// TIA Portal V19 export
FUNCTION_BLOCK "Pu_Entl.GP0x"   // FB1009, LAD
TITLE = Pumpe Abpumpen Sump
{ S7_Optimized_Access := 'TRUE' }
// Funktionen:  Entleeren /  Spülen
// stored: AutoNumber false, MemoryReserve 100, SetENOAutomatically false
   VAR RETAIN
      In { ExternalAccessible := 'False'; ExternalVisible := 'False'; ExternalWritable := 'False'} : Struct
         Auto : Bool;   // Paneltaste
         Ein : Bool;   // Paneltaste
         Leckage_ok : Bool;
         Frg_Niv_CM05 : Bool;
         Betriebsart : USInt := 0;   // Paneltaste
      END_STRUCT;
      Param { ExternalAccessible := 'False'; ExternalVisible := 'False'; ExternalWritable := 'False'} : Struct
         Spülzeit : Time;
      END_STRUCT;
      Zst { ExternalAccessible := 'False'; ExternalVisible := 'False'; ExternalWritable := 'False'} : Struct
         Niveau : USInt;
         Status_GP0x : USInt;
         Restzeit_Spülen : Time;
         TON_Spülventil_auf : Bool;
         Spuelen : Bool;
         Abpumpen : Bool;
         Bedienung_Erlaubt : Bool;
      END_STRUCT;
      Mld { ExternalAccessible := 'False'; ExternalVisible := 'False'; ExternalWritable := 'False'} : Struct
         Leckage : Bool;
         Niv_Sensorfehler : Bool;
         n_Auto : Bool;
      END_STRUCT;
      Out { ExternalAccessible := 'False'; ExternalVisible := 'False'; ExternalWritable := 'False'} : Struct
         GP0x_Ein : Bool;
         Spülventil : Bool;
      END_STRUCT;
   END_VAR
   VAR
      IEC_Timer { ExternalAccessible := 'False'; ExternalVisible := 'False'; ExternalWritable := 'False'} : Struct
         Leckage_ok { S7_SetPoint := 'True'} : TON_TIME;
         Spülventil_auf { S7_SetPoint := 'True'} : TON_TIME;
         Spülen { S7_SetPoint := 'True'} : TP_TIME;
         Leckage_niO { S7_SetPoint := 'True'} : TON_TIME;
      END_STRUCT;
      R_TRIG_Hand_EIN { ExternalAccessible := 'False'; ExternalVisible := 'False'; ExternalWritable := 'False'} : R_TRIG;
   END_VAR
   VAR_TEMP
      Spülzeit : Time;
      Leckage_ok_verz : Bool;
      posFl_Hand : Bool;
   END_VAR
   VAR CONSTANT
      Niv_TLS : USInt := 2;
      Niv_Min : USInt := 2;
      Niv_max : USInt := 20;
      Zeit_Ventil_auf : Time := T#1s;
   END_VAR
BEGIN

REGION Network 1 (SCL): Input
   // Panelbedienung und Sensoren --> Input()
   // Leckage o.k. verzögert
   #IEC_Timer.Leckage_ok(IN := #In.Leckage_ok,
                         PT := T#120s,
                         Q => #Leckage_ok_verz);

   // Timer Spülventil AUF
   #IEC_Timer.Spülventil_auf(IN := #Out.Spülventil,
                              PT := #Zeit_Ventil_auf,
                              Q => #Zst.TON_Spülventil_auf);

    // positive Flanke "Hand Ein"
   #R_TRIG_Hand_EIN(CLK := #In.Ein,
                    Q => #posFl_Hand);

   #IEC_Timer.Spülen(IN := #posFl_Hand AND #In.Betriebsart = 1,
                     PT := #Param.Spülzeit,
                     Q => #Zst.Spuelen,
                     ET => #Spülzeit);
END_REGION

REGION Network 2 (SCL): Ansteuerung
   // Zielbehälter nicht voll
   IF #In.Frg_Niv_CM05 THEN
       CASE #In.Betriebsart OF
           0:  // Entleeren

               // Spülventil zu
               #Out.Spülventil := FALSE;
               #Zst.Restzeit_Spülen := T#0s;

               // Wenn Leckage oder einmalig per Hand
               IF #In.Auto AND NOT #In.Leckage_ok OR #posFl_Hand THEN
                   #Zst.Abpumpen := TRUE;
               ELSIF #Leckage_ok_verz THEN
                   #Zst.Abpumpen := FALSE;
               END_IF;

           1: // Spülen - nur Hand
               IF #In.Ein THEN
                   IF #posFl_Hand THEN
                       #Out.Spülventil := TRUE;
                   ELSIF NOT #Zst.Spuelen AND #Zst.TON_Spülventil_auf THEN
                       #Out.Spülventil := FALSE;
                   END_IF;
                   #Zst.Restzeit_Spülen := #Param.Spülzeit - #Spülzeit;
               ELSE
                   #Zst.Spuelen := FALSE;
                   #Out.Spülventil := FALSE;
                   #Zst.Restzeit_Spülen := T#0s;
               END_IF;

               // Wenn Leckage 
               IF #Leckage_ok_verz OR (NOT #In.Auto AND NOT #In.Ein) THEN
                   #Zst.Abpumpen := FALSE;
               ELSIF NOT #In.Leckage_ok THEN
                   #Zst.Abpumpen := TRUE;
               END_IF;
       END_CASE;

       // Pumpe an    
       #Out.GP0x_Ein := #Zst.Abpumpen AND (#In.Auto OR #In.Ein);
   ELSE
       #Out.Spülventil := FALSE;
       #Zst.Restzeit_Spülen := T#0s;
       #Out.GP0x_Ein := FALSE;
   END_IF;
END_REGION

REGION Network 3 (SCL): Überwachung / Meldungen

   // Meldung Leckage verzögert
   #IEC_Timer.Leckage_niO(IN := NOT #In.Leckage_ok,
                   PT := T#30s,
                   Q => #Mld.Leckage);

   // nicht in Automatik
   #Mld.n_Auto := NOT #In.Auto AND "DB_ANLAGE".BA.Automat_ein;
END_REGION

REGION Network 4 (SCL): --> Visu
   // Status Pumpe
   "Status_E0A"(Hand := #In.Ein,
                Auto := #In.Auto,
                SonderModus_PumpeSpuelen:=FALSE,
                Stoerung := FALSE,
                Ausgang := #Out.GP0x_Ein,
                StatusByte => #Zst.Status_GP0x);
   // Anzeige Füllstand
   "Niv_Visu"(Niv_1 := TRUE,
              Niv_2 := NOT #In.Leckage_ok,
              Niv_3 := FALSE,
              Niv_4 := FALSE,
              Niv_5 := FALSE,
              Niv_6 := FALSE,
              Wert_1 := #Niv_Min,
              Wert_2 := #Niv_max,
              Wert_3 := 0,
              Wert_4 := 0,
              Wert_5 := 0,
              Wert_6 := 0,
              Niveau => #Zst.Niveau,
              Niv_Err => #Mld.Niv_Sensorfehler);

   #Zst.Bedienung_Erlaubt := NOT #In.Ein AND NOT #In.Auto;
END_REGION
END_FUNCTION_BLOCK
